(* PLC project v0.6.02_RefactorGateAndTest.project, CODESYS CODESYS V3.5 SP19 Patch 1 *)
(* stored: creationDateTime 2026-08-11T14:02:33.680684, modificationDateTime 2026-08-11T14:02:33.680684 *)

TYPE ST_PreflightHMI : STRUCT
  BtnRun : BOOL;
  PreflightOk : BOOL;
  PreflightDone : BOOL;
  PreflightBusy : BOOL;
  PreflightErrorId : WORD;
END_STRUCT;
END_TYPE
